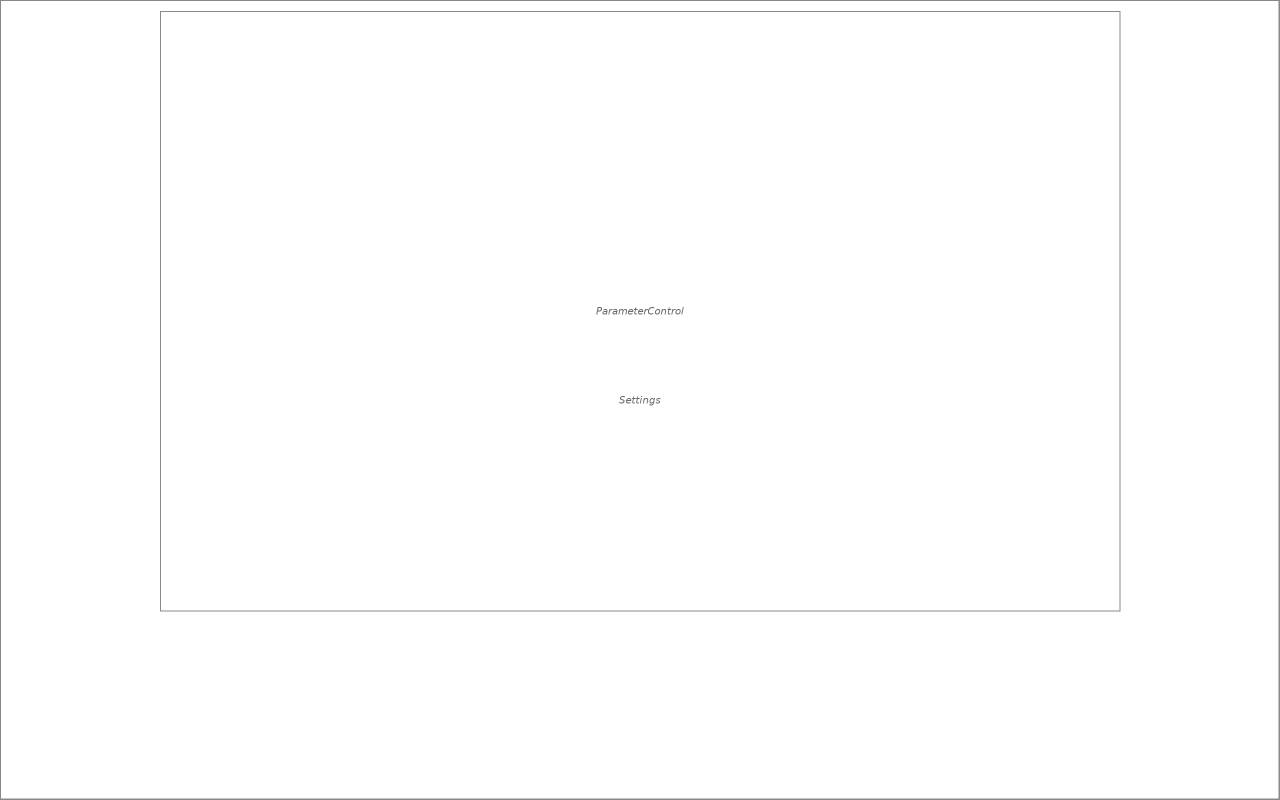
VISUALIZATION ParameterScreen  // 1280x800, background image BackGroundImagePool_SVG.Background_Sides
VAR_IN_OUT
	bCmdParameter : BOOL ; // Go to parameter screen
	nUnitsProduced : UDINT ; // Units produced in machine lifetime
END_VAR
    Frame (0,0 1280x800)
        shows Settings(bCmdParameter := bCmdParameter, nUnitsProduced := nUnitsProduced)
    Frame (160,11 960x600)
        shows ParameterControl()
END_VISUALIZATION

(* stored: Version 1.1.0.1, ProductVersion 3.1.4024.9
   Visu ParameterScreen: Id {be090142-cc46-445b-bfe3-261de64e9afe} *)
